SUBAPPLICATION Uebung_087a2 (* Beispiel für E_DEMUX_4 *)
  (* Standard: 61499-2; Description: Copyright (c) 2023 Meisterschulen am Ostbahnhof This program and the accompanying materials are made available under the terms of the Eclipse Public License 2.0 which is available at https://www.eclipse.org/legal/epl-2.0/ SPDX-License-Identifier: EPL-2.0 Beispiel für E_CTD Aufwärts zählen UAO Curriculum Module 3 - The IEC 61499 Standard, Seite 93 *)
  (* Version 1.0, 2023-10-23, Franz Höpfinger, Meisterschulen am Ostbahnhof *)
  PACKAGE Uebungen;
  IMPORT logiBUS::io::DI::logiBUS_DI::Input_I1;
  IMPORT logiBUS::io::DI::logiBUS_DI::Input_I2;
  IMPORT logiBUS::io::DI::logiBUS_DI::Input_I3;
  IMPORT logiBUS::io::DI::logiBUS_DI::Input_I4;
  IMPORT logiBUS::io::DQ::logiBUS_DO::Output_Q1;
  IMPORT logiBUS::io::DQ::logiBUS_DO::Output_Q2;
  IMPORT logiBUS::io::DQ::logiBUS_DO::Output_Q3;
  IMPORT logiBUS::io::DQ::logiBUS_DO::Output_Q4;
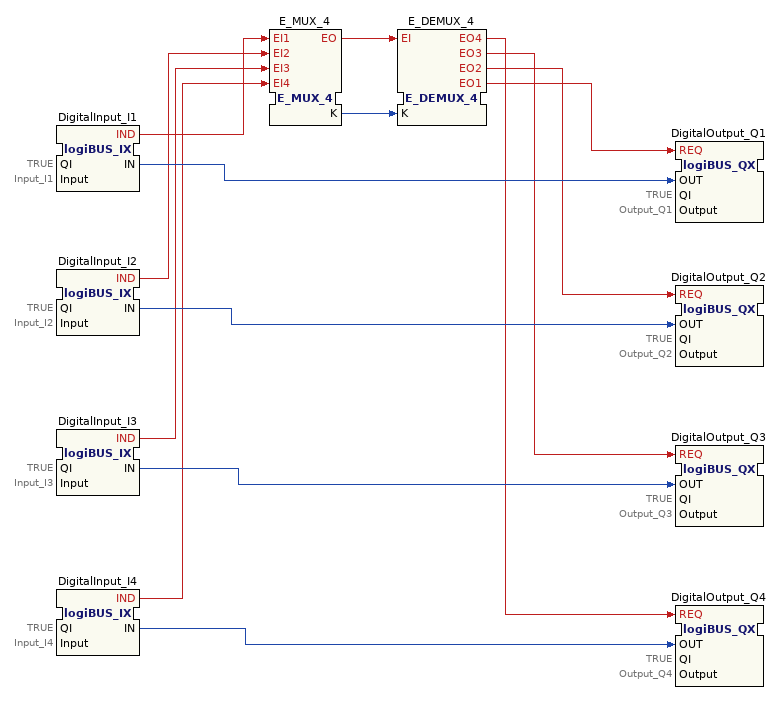
  FBS
    DigitalOutput_Q1 : logiBUS::io::DQ::logiBUS_QX(QI := TRUE, Output := Output_Q1);
    DigitalInput_I1 : logiBUS::io::DI::logiBUS_IX(QI := TRUE, Input := Input_I1);
    DigitalOutput_Q2 : logiBUS::io::DQ::logiBUS_QX(QI := TRUE, Output := Output_Q2);
    DigitalInput_I2 : logiBUS::io::DI::logiBUS_IX(QI := TRUE, Input := Input_I2);
    DigitalOutput_Q3 : logiBUS::io::DQ::logiBUS_QX(QI := TRUE, Output := Output_Q3);
    DigitalInput_I3 : logiBUS::io::DI::logiBUS_IX(QI := TRUE, Input := Input_I3);
    DigitalOutput_Q4 : logiBUS::io::DQ::logiBUS_QX(QI := TRUE, Output := Output_Q4);
    DigitalInput_I4 : logiBUS::io::DI::logiBUS_IX(QI := TRUE, Input := Input_I4);
    E_DEMUX_4 : iec61499::events::E_DEMUX_4;
    E_MUX_4 : iec61499::events::E_MUX_4;
  END_FBS
  EVENT_CONNECTIONS
    E_MUX_4.EO TO E_DEMUX_4.EI;
    DigitalInput_I1.IND TO E_MUX_4.EI1;
    DigitalInput_I2.IND TO E_MUX_4.EI2;
    DigitalInput_I3.IND TO E_MUX_4.EI3;
    DigitalInput_I4.IND TO E_MUX_4.EI4;
    E_DEMUX_4.EO4 TO DigitalOutput_Q4.REQ;
    E_DEMUX_4.EO3 TO DigitalOutput_Q3.REQ;
    E_DEMUX_4.EO2 TO DigitalOutput_Q2.REQ;
    E_DEMUX_4.EO1 TO DigitalOutput_Q1.REQ;
  END_CONNECTIONS
  DATA_CONNECTIONS
    E_MUX_4.K TO E_DEMUX_4.K;
    DigitalInput_I1.IN TO DigitalOutput_Q1.OUT;
    DigitalInput_I2.IN TO DigitalOutput_Q2.OUT;
    DigitalInput_I3.IN TO DigitalOutput_Q3.OUT;
    DigitalInput_I4.IN TO DigitalOutput_Q4.OUT;
  END_CONNECTIONS
END_SUBAPPLICATION
